// TwinCAT 3 PLC project FMCmd
// Title: FM Cmd
// Company: FrameworkMonorepo
// ProjectVersion: 0.0.1
// ProgramVersion: 3.1.4024.0
// libraries:
//   FM Common Interfaces, * (FrameworkMonorepo)
//   Tc2_System, * (Beckhoff Automation GmbH)
//   Tc2_Utilities, * (Beckhoff Automation GmbH)
// project tree:
//   Cmd/ Cmd.TcPOU
//   Version/ Global_Version.TcGVL
// (motion and I/O tree: see PLC project fmtypes)
// real-time tasks:
//   TASK BindingTestTask: cycle T#1ms, priority 20, ADS port 350
//   TASK PlcTask: cycle T#1ms, priority 21, ADS port 351
//   TASK PlcTask1: cycle T#1ms, priority 22, ADS port 352
//   TASK PlcTask2: cycle T#1ms, priority 23, ADS port 353
//   TASK MathTestTask: cycle T#1ms, priority 24, ADS port 354
//   TASK TimesTestsTask: cycle T#1ms, priority 25, ADS port 355

// ---- Version/Global_Version.TcGVL
{attribute 'TcGenerated'}
{attribute 'no-analysis'}
{attribute 'linkalways'}
// This function has been automatically generated from the project information.
VAR_GLOBAL CONSTANT
	{attribute 'const_non_replaced'}
	stLibVersion_FM_Cmd : ST_LibVersion := (iMajor := 0, iMinor := 0, iBuild := 1, iRevision := 0, nFlags := 0, sVersion := '0.0.1');
END_VAR

// ---- Cmd/Cmd.TcPOU
FUNCTION_BLOCK Cmd IMPLEMENTS Cyclic
VAR
	startProcess : NT_StartProcess;
END_VAR

{attribute 'monitoring' := 'call'}
PROPERTY Busy : BOOL
GET
Busy := startProcess.BUSY;
END_GET
END_PROPERTY

METHOD Cyclic
startProcess(START := FALSE);
END_METHOD

METHOD Execute
VAR_INPUT
	command : T_MaxString;
	arguments : T_MaxString;
	workingDirectory : T_MaxString;
END_VAR
startProcess(
	DIRNAME := workingDirectory,
	PATHSTR := command,
	COMNDLINE := arguments,
	START := TRUE
);
END_METHOD

END_FUNCTION_BLOCK
